// TIA Portal V16 export
// export: Created 2024-03-27T10:04:38.8710703Z, ExportSetting WithDefaults, DisplayName Totally Integrated Automation Portal, DisplayVersion V16, DisplayName TIA Portal Version Control Interface, DisplayVersion V16, DisplayName TIA Portal Openness, DisplayVersion V16, DisplayName STEP 7 Professional, DisplayVersion V16, DisplayName STEP 7 Safety, DisplayVersion V16, DisplayName WinCC Advanced, DisplayVersion V16
TYPE "UR_4_T2O_TCP"
// stored: IsFailsafeCompliant false
   STRUCT
      "TCP Position (X,Y,Z) [m]" : Array[0..2] of Real;
      "TCP Position (RX,RY,RZ) [rad]" : Array[0..2] of Real;
      "TCP velocity (X,Y,Z) [m/s]" : Array[0..2] of Real;
      "TCP velocity (RX,RY,RZ) [rad/s]" : Array[0..2] of Real;
      "TCP force (X,Y,Z) [N]" : Array[0..2] of Real;
      "TCP torque (X,Y,Z) [Nm]" : Array[0..2] of Real;
      "TCP force scalar [N]" : Real;
   END_STRUCT;
END_TYPE
